// TIA Portal V18 export
FUNCTION_BLOCK "ST10_CountCycleTimeMain"   // FB1009, LAD
{ S7_Optimized_Access := 'TRUE' }
VERSION : 0.1
// stored: AutoNumber false, IsIECCheckEnabled false, IsRetainMemResEnabled false, MemoryReserve 100, SetENOAutomatically false, UDAEnableTagReadback false
   VAR_INPUT
      iAlwaysOn : Bool;
      iRun : Bool;
      iManualMode : Bool;
      iAutoMode : Bool;
      iAutoRunning : Bool;
   END_VAR
   VAR
      MianCountCycleTime { S7_SetPoint := 'True'} : "Count_CycleTime";
      PM1CountCycleTime { S7_SetPoint := 'True'} : "Count_CycleTime_V3";
      PM2CountCycleTime { S7_SetPoint := 'True'} : "Count_CycleTime_V3";
      PM3CountCycleTime { S7_SetPoint := 'True'} : "Count_CycleTime_V3";
      PM4CountCycleTime { S7_SetPoint := 'True'} : "Count_CycleTime_V3";
      PM5CountCycleTime { S7_SetPoint := 'True'} : "Count_CycleTime_V3";
      PM6CountCycleTime { S7_SetPoint := 'True'} : "Count_CycleTime_V3";
      PM7CountCycleTime { S7_SetPoint := 'True'} : "Count_CycleTime_V3";
      PM8CountCycleTime { S7_SetPoint := 'True'} : "Count_CycleTime_V3";
      PM9CountCycleTime { S7_SetPoint := 'True'} : "Count_CycleTime_V3";
      PM10CountCycleTime { S7_SetPoint := 'True'} : "Count_CycleTime_V3";
      PM11CountCycleTime { S7_SetPoint := 'True'} : "Count_CycleTime_V3";
      PM12CountCycleTime { S7_SetPoint := 'True'} : "Count_CycleTime_V3";
      PM13CountCycleTime { S7_SetPoint := 'True'} : "Count_CycleTime_V3";
      PM14CountCycleTime { S7_SetPoint := 'True'} : "Count_CycleTime_V3";
      PM15CountCycleTime { S7_SetPoint := 'True'} : "Count_CycleTime_V3";
      PM16CountCycleTime { S7_SetPoint := 'True'} : "Count_CycleTime_V3";
      PM17CountCycleTime { S7_SetPoint := 'True'} : "Count_CycleTime_V3";
      PM18CountCycleTime { S7_SetPoint := 'True'} : "Count_CycleTime_V3";
      PM19CountCycleTime { S7_SetPoint := 'True'} : "Count_CycleTime_V3";
      PM20CountCycleTime { S7_SetPoint := 'True'} : "Count_CycleTime_V3";
      PM21CountCycleTime { S7_SetPoint := 'True'} : "Count_CycleTime_V3";
      PM22CountCycleTime { S7_SetPoint := 'True'} : "Count_CycleTime_V3";
      PM23CountCycleTime { S7_SetPoint := 'True'} : "Count_CycleTime_V3";
      PM24CountCycleTime { S7_SetPoint := 'True'} : "Count_CycleTime_V3";
      PM25CountCycleTime { S7_SetPoint := 'True'} : "Count_CycleTime_V3";
      PM26CountCycleTime { S7_SetPoint := 'True'} : "Count_CycleTime_V3";
      PM27CountCycleTime { S7_SetPoint := 'True'} : "Count_CycleTime_V3";
      PM28CountCycleTime { S7_SetPoint := 'True'} : "Count_CycleTime_V3";
      PM29CountCycleTime { S7_SetPoint := 'True'} : "Count_CycleTime_V3";
      PM30CountCycleTime { S7_SetPoint := 'True'} : "Count_CycleTime_V3";
   END_VAR
BEGIN

REGION Network 1: Mian Count & CycleTime
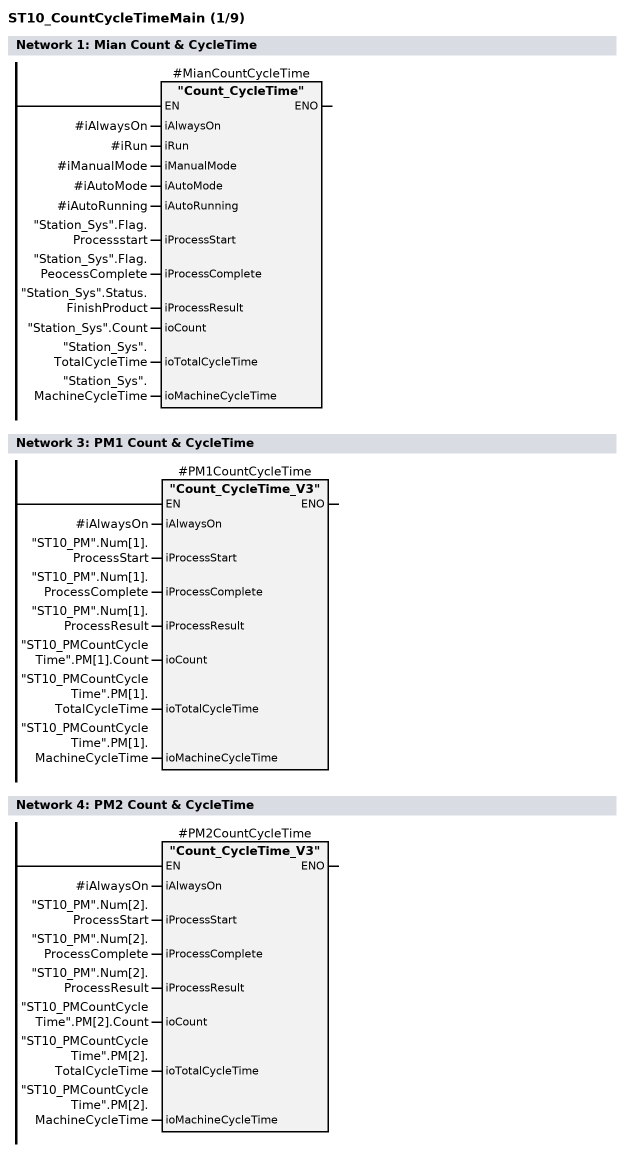
   RUNG wire#powerrail
      #MianCountCycleTime(iAlwaysOn := #iAlwaysOn, iRun := #iRun, iManualMode := #iManualMode, iAutoMode := #iAutoMode, iAutoRunning := #iAutoRunning, iProcessStart := "Station_Sys".Flag.Processstart, iProcessComplete := "Station_Sys".Flag.PeocessComplete, iProcessResult := "Station_Sys".Status.FinishProduct, ioCount := "Station_Sys".Count, ioTotalCycleTime := "Station_Sys".TotalCycleTime, ioMachineCycleTime := "Station_Sys".MachineCycleTime)
   END_RUNG
   // the same network as SCL:
   #MianCountCycleTime(iAlwaysOn := #iAlwaysOn,   // "Count_CycleTime"
                       iRun := #iRun,
                       iManualMode := #iManualMode,
                       iAutoMode := #iAutoMode,
                       iAutoRunning := #iAutoRunning,
                       iProcessStart := "Station_Sys".Flag.Processstart,
                       iProcessComplete := "Station_Sys".Flag.PeocessComplete,
                       iProcessResult := "Station_Sys".Status.FinishProduct,
                       ioCount := "Station_Sys".Count,
                       ioTotalCycleTime := "Station_Sys".TotalCycleTime,
                       ioMachineCycleTime := "Station_Sys".MachineCycleTime);
END_REGION

REGION Network 2 (SCL)
   "ST10_PMCountCycleTime".PM[1].Num := 1;
   "ST10_PMCountCycleTime".PM[2].Num := 2;
   "ST10_PMCountCycleTime".PM[3].Num := 3;
   "ST10_PMCountCycleTime".PM[4].Num := 4;
   "ST10_PMCountCycleTime".PM[5].Num := 5;
   "ST10_PMCountCycleTime".PM[6].Num := 6;
   "ST10_PMCountCycleTime".PM[7].Num := 7;
   "ST10_PMCountCycleTime".PM[8].Num := 8;
   "ST10_PMCountCycleTime".PM[9].Num := 9;
   "ST10_PMCountCycleTime".PM[10].Num := 10;
   "ST10_PMCountCycleTime".PM[11].Num := 11;
   "ST10_PMCountCycleTime".PM[12].Num := 12;
   "ST10_PMCountCycleTime".PM[13].Num := 13;
   "ST10_PMCountCycleTime".PM[14].Num := 14;
   "ST10_PMCountCycleTime".PM[15].Num := 15;
   "ST10_PMCountCycleTime".PM[16].Num := 16;
   "ST10_PMCountCycleTime".PM[17].Num := 17;
   "ST10_PMCountCycleTime".PM[18].Num := 18;
   "ST10_PMCountCycleTime".PM[19].Num := 19;
   "ST10_PMCountCycleTime".PM[20].Num := 20;
   "ST10_PMCountCycleTime".PM[21].Num := 21;
   "ST10_PMCountCycleTime".PM[22].Num := 22;
   "ST10_PMCountCycleTime".PM[23].Num := 23;
   "ST10_PMCountCycleTime".PM[24].Num := 24;
   "ST10_PMCountCycleTime".PM[25].Num := 25;
   // "ST70_PMCountCycleTime".PM[5].Num := 5;
   // "ST70_PMCountCycleTime".PM[6].Num := 6;
   // "ST70_PMCountCycleTime".PM[7].Num := 7;
   // "ST70_PMCountCycleTime".PM[8].Num := 8;
   // "ST70_PMCountCycleTime".PM[9].Num := 9;
   // "ST70_PMCountCycleTime".PM[10].Num := 10;
   //TEST
   (*
   "ST10_PMCountCycleTime".PM[1].Count.OK[0] := 10;
   "ST10_PMCountCycleTime".PM[2].Count.OK[0] := 20;
   "ST10_PMCountCycleTime".PM[3].Count.OK[0] := 30;
   "ST10_PMCountCycleTime".PM[4].Count.OK[0] := 40;
   "ST10_PMCountCycleTime".PM[5].Count.OK[0] := 50;
   "ST10_PMCountCycleTime".PM[6].Count.OK[0] := 60;
   "ST10_PMCountCycleTime".PM[7].Count.OK[0] := 70;
   "ST10_PMCountCycleTime".PM[8].Count.OK[0] := 80;
   "ST10_PMCountCycleTime".PM[9].Count.OK[0] := 90;
   "ST10_PMCountCycleTime".PM[10].Count.OK[0] := 100;

   "ST10_PMCountCycleTime".PM[1].TotalCycleTime.No[0] := 100;
   "ST10_PMCountCycleTime".PM[2].TotalCycleTime.No[0] := 200;
   "ST10_PMCountCycleTime".PM[3].TotalCycleTime.No[0] := 300;
   "ST10_PMCountCycleTime".PM[4].TotalCycleTime.No[0] := 400;
   "ST10_PMCountCycleTime".PM[5].TotalCycleTime.No[0] := 500;
   "ST10_PMCountCycleTime".PM[6].TotalCycleTime.No[0] := 600;
   "ST10_PMCountCycleTime".PM[7].TotalCycleTime.No[0] := 700;
   "ST10_PMCountCycleTime".PM[8].TotalCycleTime.No[0] := 800;
   "ST10_PMCountCycleTime".PM[9].TotalCycleTime.No[0] := 900;
   "ST10_PMCountCycleTime".PM[10].TotalCycleTime.No[0] := 1000;

   "ST10_PMCountCycleTime".PM[1].MachineCycleTime.No[0] := 110;
   "ST10_PMCountCycleTime".PM[2].MachineCycleTime.No[0] := 220;
   "ST10_PMCountCycleTime".PM[3].MachineCycleTime.No[0] := 330;
   "ST10_PMCountCycleTime".PM[4].MachineCycleTime.No[0] := 440;
   "ST10_PMCountCycleTime".PM[5].MachineCycleTime.No[0] := 550;
   "ST10_PMCountCycleTime".PM[6].MachineCycleTime.No[0] := 660;
   "ST10_PMCountCycleTime".PM[7].MachineCycleTime.No[0] := 770;
   "ST10_PMCountCycleTime".PM[8].MachineCycleTime.No[0] := 880;
   "ST10_PMCountCycleTime".PM[9].MachineCycleTime.No[0] := 990;
   "ST10_PMCountCycleTime".PM[10].MachineCycleTime.No[0] := 1010;
   *)
END_REGION

REGION Network 3: PM1 Count & CycleTime
   RUNG wire#powerrail
      #PM1CountCycleTime(iAlwaysOn := #iAlwaysOn, iProcessStart := "ST10_PM".Num[1].ProcessStart, iProcessComplete := "ST10_PM".Num[1].ProcessComplete, iProcessResult := "ST10_PM".Num[1].ProcessResult, ioCount := "ST10_PMCountCycleTime".PM[1].Count, ioTotalCycleTime := "ST10_PMCountCycleTime".PM[1].TotalCycleTime, ioMachineCycleTime := "ST10_PMCountCycleTime".PM[1].MachineCycleTime)
   END_RUNG
   // the same network as SCL:
   #PM1CountCycleTime(iAlwaysOn := #iAlwaysOn,   // "Count_CycleTime_V3"
                      iProcessStart := "ST10_PM".Num[1].ProcessStart,
                      iProcessComplete := "ST10_PM".Num[1].ProcessComplete,
                      iProcessResult := "ST10_PM".Num[1].ProcessResult,
                      ioCount := "ST10_PMCountCycleTime".PM[1].Count,
                      ioTotalCycleTime := "ST10_PMCountCycleTime".PM[1].TotalCycleTime,
                      ioMachineCycleTime := "ST10_PMCountCycleTime".PM[1].MachineCycleTime);
END_REGION

REGION Network 4: PM2 Count & CycleTime
   RUNG wire#powerrail
      #PM2CountCycleTime(iAlwaysOn := #iAlwaysOn, iProcessStart := "ST10_PM".Num[2].ProcessStart, iProcessComplete := "ST10_PM".Num[2].ProcessComplete, iProcessResult := "ST10_PM".Num[2].ProcessResult, ioCount := "ST10_PMCountCycleTime".PM[2].Count, ioTotalCycleTime := "ST10_PMCountCycleTime".PM[2].TotalCycleTime, ioMachineCycleTime := "ST10_PMCountCycleTime".PM[2].MachineCycleTime)
   END_RUNG
   // the same network as SCL:
   #PM2CountCycleTime(iAlwaysOn := #iAlwaysOn,   // "Count_CycleTime_V3"
                      iProcessStart := "ST10_PM".Num[2].ProcessStart,
                      iProcessComplete := "ST10_PM".Num[2].ProcessComplete,
                      iProcessResult := "ST10_PM".Num[2].ProcessResult,
                      ioCount := "ST10_PMCountCycleTime".PM[2].Count,
                      ioTotalCycleTime := "ST10_PMCountCycleTime".PM[2].TotalCycleTime,
                      ioMachineCycleTime := "ST10_PMCountCycleTime".PM[2].MachineCycleTime);
END_REGION

REGION Network 5: PM3 Count & CycleTime
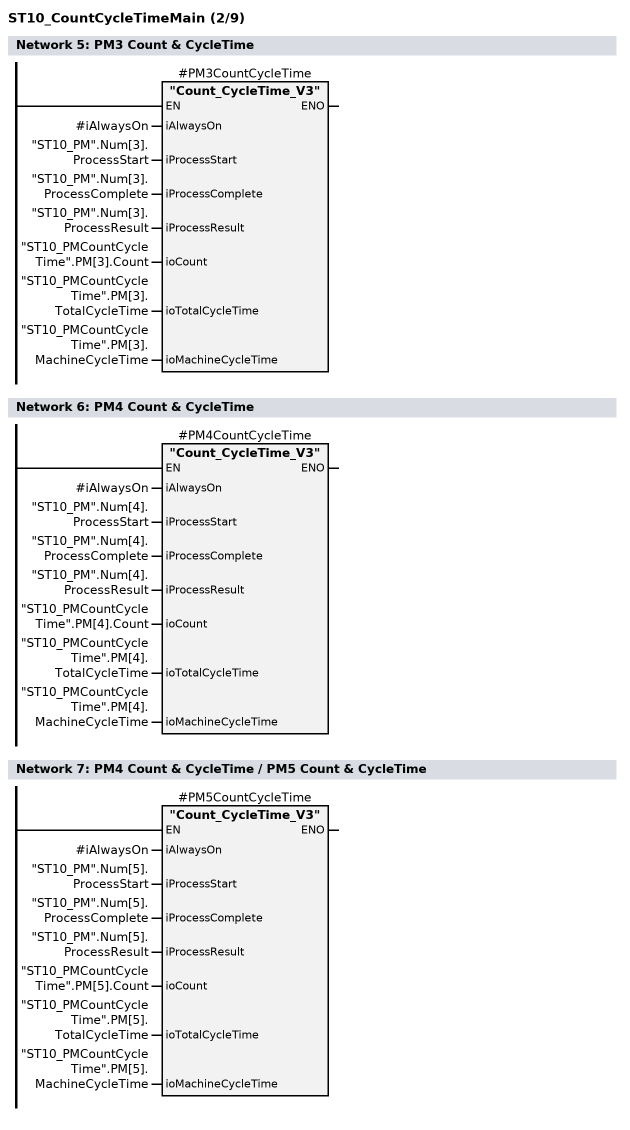
   RUNG wire#powerrail
      #PM3CountCycleTime(iAlwaysOn := #iAlwaysOn, iProcessStart := "ST10_PM".Num[3].ProcessStart, iProcessComplete := "ST10_PM".Num[3].ProcessComplete, iProcessResult := "ST10_PM".Num[3].ProcessResult, ioCount := "ST10_PMCountCycleTime".PM[3].Count, ioTotalCycleTime := "ST10_PMCountCycleTime".PM[3].TotalCycleTime, ioMachineCycleTime := "ST10_PMCountCycleTime".PM[3].MachineCycleTime)
   END_RUNG
   // the same network as SCL:
   #PM3CountCycleTime(iAlwaysOn := #iAlwaysOn,   // "Count_CycleTime_V3"
                      iProcessStart := "ST10_PM".Num[3].ProcessStart,
                      iProcessComplete := "ST10_PM".Num[3].ProcessComplete,
                      iProcessResult := "ST10_PM".Num[3].ProcessResult,
                      ioCount := "ST10_PMCountCycleTime".PM[3].Count,
                      ioTotalCycleTime := "ST10_PMCountCycleTime".PM[3].TotalCycleTime,
                      ioMachineCycleTime := "ST10_PMCountCycleTime".PM[3].MachineCycleTime);
END_REGION

REGION Network 6: PM4 Count & CycleTime
   RUNG wire#powerrail
      #PM4CountCycleTime(iAlwaysOn := #iAlwaysOn, iProcessStart := "ST10_PM".Num[4].ProcessStart, iProcessComplete := "ST10_PM".Num[4].ProcessComplete, iProcessResult := "ST10_PM".Num[4].ProcessResult, ioCount := "ST10_PMCountCycleTime".PM[4].Count, ioTotalCycleTime := "ST10_PMCountCycleTime".PM[4].TotalCycleTime, ioMachineCycleTime := "ST10_PMCountCycleTime".PM[4].MachineCycleTime)
   END_RUNG
   // the same network as SCL:
   #PM4CountCycleTime(iAlwaysOn := #iAlwaysOn,   // "Count_CycleTime_V3"
                      iProcessStart := "ST10_PM".Num[4].ProcessStart,
                      iProcessComplete := "ST10_PM".Num[4].ProcessComplete,
                      iProcessResult := "ST10_PM".Num[4].ProcessResult,
                      ioCount := "ST10_PMCountCycleTime".PM[4].Count,
                      ioTotalCycleTime := "ST10_PMCountCycleTime".PM[4].TotalCycleTime,
                      ioMachineCycleTime := "ST10_PMCountCycleTime".PM[4].MachineCycleTime);
END_REGION

REGION Network 7: PM4 Count & CycleTime / PM5 Count & CycleTime
   RUNG wire#powerrail
      #PM5CountCycleTime(iAlwaysOn := #iAlwaysOn, iProcessStart := "ST10_PM".Num[5].ProcessStart, iProcessComplete := "ST10_PM".Num[5].ProcessComplete, iProcessResult := "ST10_PM".Num[5].ProcessResult, ioCount := "ST10_PMCountCycleTime".PM[5].Count, ioTotalCycleTime := "ST10_PMCountCycleTime".PM[5].TotalCycleTime, ioMachineCycleTime := "ST10_PMCountCycleTime".PM[5].MachineCycleTime)
   END_RUNG
   // the same network as SCL:
   #PM5CountCycleTime(iAlwaysOn := #iAlwaysOn,   // "Count_CycleTime_V3"
                      iProcessStart := "ST10_PM".Num[5].ProcessStart,
                      iProcessComplete := "ST10_PM".Num[5].ProcessComplete,
                      iProcessResult := "ST10_PM".Num[5].ProcessResult,
                      ioCount := "ST10_PMCountCycleTime".PM[5].Count,
                      ioTotalCycleTime := "ST10_PMCountCycleTime".PM[5].TotalCycleTime,
                      ioMachineCycleTime := "ST10_PMCountCycleTime".PM[5].MachineCycleTime);
END_REGION

REGION Network 8: PM4 Count & CycleTime / PM6 Count & CycleTime
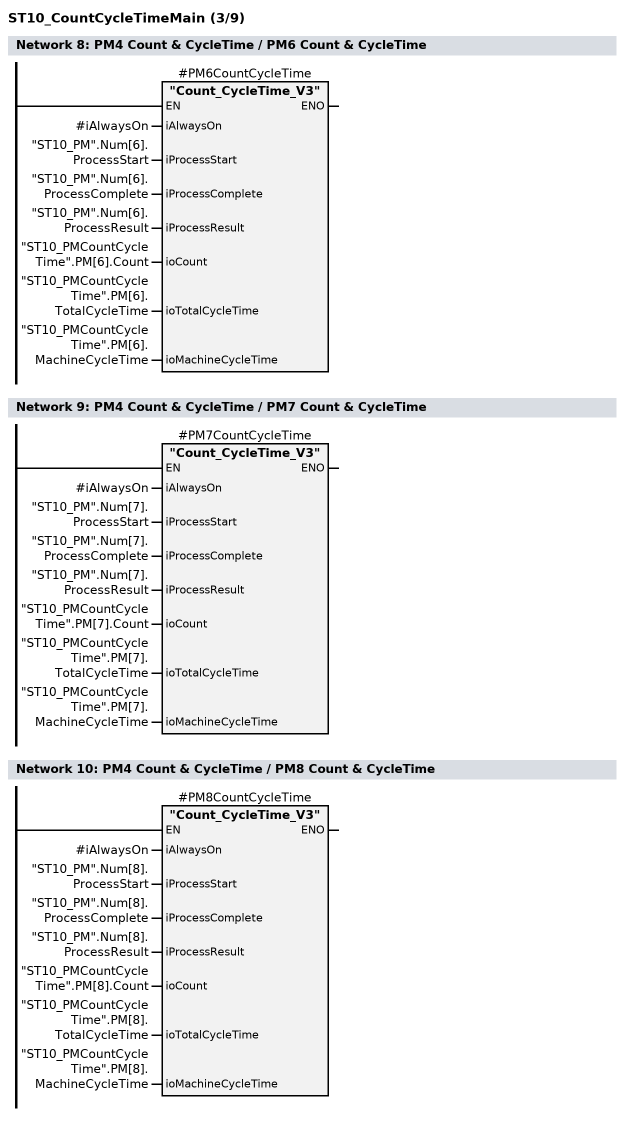
   RUNG wire#powerrail
      #PM6CountCycleTime(iAlwaysOn := #iAlwaysOn, iProcessStart := "ST10_PM".Num[6].ProcessStart, iProcessComplete := "ST10_PM".Num[6].ProcessComplete, iProcessResult := "ST10_PM".Num[6].ProcessResult, ioCount := "ST10_PMCountCycleTime".PM[6].Count, ioTotalCycleTime := "ST10_PMCountCycleTime".PM[6].TotalCycleTime, ioMachineCycleTime := "ST10_PMCountCycleTime".PM[6].MachineCycleTime)
   END_RUNG
   // the same network as SCL:
   #PM6CountCycleTime(iAlwaysOn := #iAlwaysOn,   // "Count_CycleTime_V3"
                      iProcessStart := "ST10_PM".Num[6].ProcessStart,
                      iProcessComplete := "ST10_PM".Num[6].ProcessComplete,
                      iProcessResult := "ST10_PM".Num[6].ProcessResult,
                      ioCount := "ST10_PMCountCycleTime".PM[6].Count,
                      ioTotalCycleTime := "ST10_PMCountCycleTime".PM[6].TotalCycleTime,
                      ioMachineCycleTime := "ST10_PMCountCycleTime".PM[6].MachineCycleTime);
END_REGION

REGION Network 9: PM4 Count & CycleTime / PM7 Count & CycleTime
   RUNG wire#powerrail
      #PM7CountCycleTime(iAlwaysOn := #iAlwaysOn, iProcessStart := "ST10_PM".Num[7].ProcessStart, iProcessComplete := "ST10_PM".Num[7].ProcessComplete, iProcessResult := "ST10_PM".Num[7].ProcessResult, ioCount := "ST10_PMCountCycleTime".PM[7].Count, ioTotalCycleTime := "ST10_PMCountCycleTime".PM[7].TotalCycleTime, ioMachineCycleTime := "ST10_PMCountCycleTime".PM[7].MachineCycleTime)
   END_RUNG
   // the same network as SCL:
   #PM7CountCycleTime(iAlwaysOn := #iAlwaysOn,   // "Count_CycleTime_V3"
                      iProcessStart := "ST10_PM".Num[7].ProcessStart,
                      iProcessComplete := "ST10_PM".Num[7].ProcessComplete,
                      iProcessResult := "ST10_PM".Num[7].ProcessResult,
                      ioCount := "ST10_PMCountCycleTime".PM[7].Count,
                      ioTotalCycleTime := "ST10_PMCountCycleTime".PM[7].TotalCycleTime,
                      ioMachineCycleTime := "ST10_PMCountCycleTime".PM[7].MachineCycleTime);
END_REGION

REGION Network 10: PM4 Count & CycleTime / PM8 Count & CycleTime
   RUNG wire#powerrail
      #PM8CountCycleTime(iAlwaysOn := #iAlwaysOn, iProcessStart := "ST10_PM".Num[8].ProcessStart, iProcessComplete := "ST10_PM".Num[8].ProcessComplete, iProcessResult := "ST10_PM".Num[8].ProcessResult, ioCount := "ST10_PMCountCycleTime".PM[8].Count, ioTotalCycleTime := "ST10_PMCountCycleTime".PM[8].TotalCycleTime, ioMachineCycleTime := "ST10_PMCountCycleTime".PM[8].MachineCycleTime)
   END_RUNG
   // the same network as SCL:
   #PM8CountCycleTime(iAlwaysOn := #iAlwaysOn,   // "Count_CycleTime_V3"
                      iProcessStart := "ST10_PM".Num[8].ProcessStart,
                      iProcessComplete := "ST10_PM".Num[8].ProcessComplete,
                      iProcessResult := "ST10_PM".Num[8].ProcessResult,
                      ioCount := "ST10_PMCountCycleTime".PM[8].Count,
                      ioTotalCycleTime := "ST10_PMCountCycleTime".PM[8].TotalCycleTime,
                      ioMachineCycleTime := "ST10_PMCountCycleTime".PM[8].MachineCycleTime);
END_REGION

REGION Network 11: PM4 Count & CycleTime / PM9 Count & CycleTime
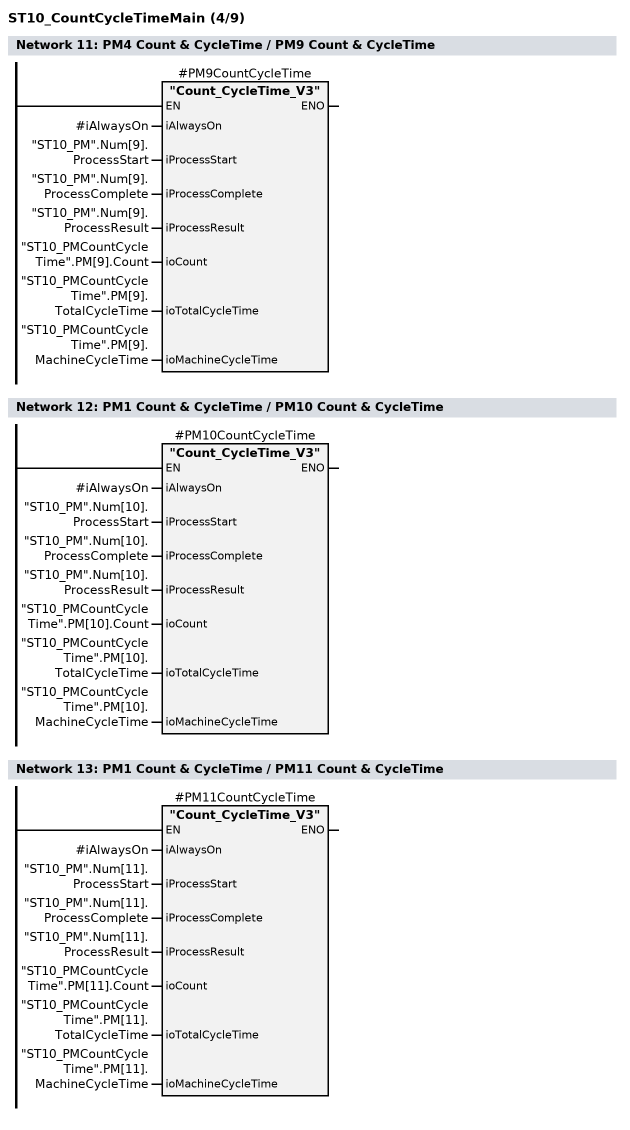
   RUNG wire#powerrail
      #PM9CountCycleTime(iAlwaysOn := #iAlwaysOn, iProcessStart := "ST10_PM".Num[9].ProcessStart, iProcessComplete := "ST10_PM".Num[9].ProcessComplete, iProcessResult := "ST10_PM".Num[9].ProcessResult, ioCount := "ST10_PMCountCycleTime".PM[9].Count, ioTotalCycleTime := "ST10_PMCountCycleTime".PM[9].TotalCycleTime, ioMachineCycleTime := "ST10_PMCountCycleTime".PM[9].MachineCycleTime)
   END_RUNG
   // the same network as SCL:
   #PM9CountCycleTime(iAlwaysOn := #iAlwaysOn,   // "Count_CycleTime_V3"
                      iProcessStart := "ST10_PM".Num[9].ProcessStart,
                      iProcessComplete := "ST10_PM".Num[9].ProcessComplete,
                      iProcessResult := "ST10_PM".Num[9].ProcessResult,
                      ioCount := "ST10_PMCountCycleTime".PM[9].Count,
                      ioTotalCycleTime := "ST10_PMCountCycleTime".PM[9].TotalCycleTime,
                      ioMachineCycleTime := "ST10_PMCountCycleTime".PM[9].MachineCycleTime);
END_REGION

REGION Network 12: PM1 Count & CycleTime / PM10 Count & CycleTime
   RUNG wire#powerrail
      #PM10CountCycleTime(iAlwaysOn := #iAlwaysOn, iProcessStart := "ST10_PM".Num[10].ProcessStart, iProcessComplete := "ST10_PM".Num[10].ProcessComplete, iProcessResult := "ST10_PM".Num[10].ProcessResult, ioCount := "ST10_PMCountCycleTime".PM[10].Count, ioTotalCycleTime := "ST10_PMCountCycleTime".PM[10].TotalCycleTime, ioMachineCycleTime := "ST10_PMCountCycleTime".PM[10].MachineCycleTime)
   END_RUNG
   // the same network as SCL:
   #PM10CountCycleTime(iAlwaysOn := #iAlwaysOn,   // "Count_CycleTime_V3"
                       iProcessStart := "ST10_PM".Num[10].ProcessStart,
                       iProcessComplete := "ST10_PM".Num[10].ProcessComplete,
                       iProcessResult := "ST10_PM".Num[10].ProcessResult,
                       ioCount := "ST10_PMCountCycleTime".PM[10].Count,
                       ioTotalCycleTime := "ST10_PMCountCycleTime".PM[10].TotalCycleTime,
                       ioMachineCycleTime := "ST10_PMCountCycleTime".PM[10].MachineCycleTime);
END_REGION

REGION Network 13: PM1 Count & CycleTime / PM11 Count & CycleTime
   RUNG wire#powerrail
      #PM11CountCycleTime(iAlwaysOn := #iAlwaysOn, iProcessStart := "ST10_PM".Num[11].ProcessStart, iProcessComplete := "ST10_PM".Num[11].ProcessComplete, iProcessResult := "ST10_PM".Num[11].ProcessResult, ioCount := "ST10_PMCountCycleTime".PM[11].Count, ioTotalCycleTime := "ST10_PMCountCycleTime".PM[11].TotalCycleTime, ioMachineCycleTime := "ST10_PMCountCycleTime".PM[11].MachineCycleTime)
   END_RUNG
   // the same network as SCL:
   #PM11CountCycleTime(iAlwaysOn := #iAlwaysOn,   // "Count_CycleTime_V3"
                       iProcessStart := "ST10_PM".Num[11].ProcessStart,
                       iProcessComplete := "ST10_PM".Num[11].ProcessComplete,
                       iProcessResult := "ST10_PM".Num[11].ProcessResult,
                       ioCount := "ST10_PMCountCycleTime".PM[11].Count,
                       ioTotalCycleTime := "ST10_PMCountCycleTime".PM[11].TotalCycleTime,
                       ioMachineCycleTime := "ST10_PMCountCycleTime".PM[11].MachineCycleTime);
END_REGION

REGION Network 14: PM1 Count & CycleTime / PM12 Count & CycleTime
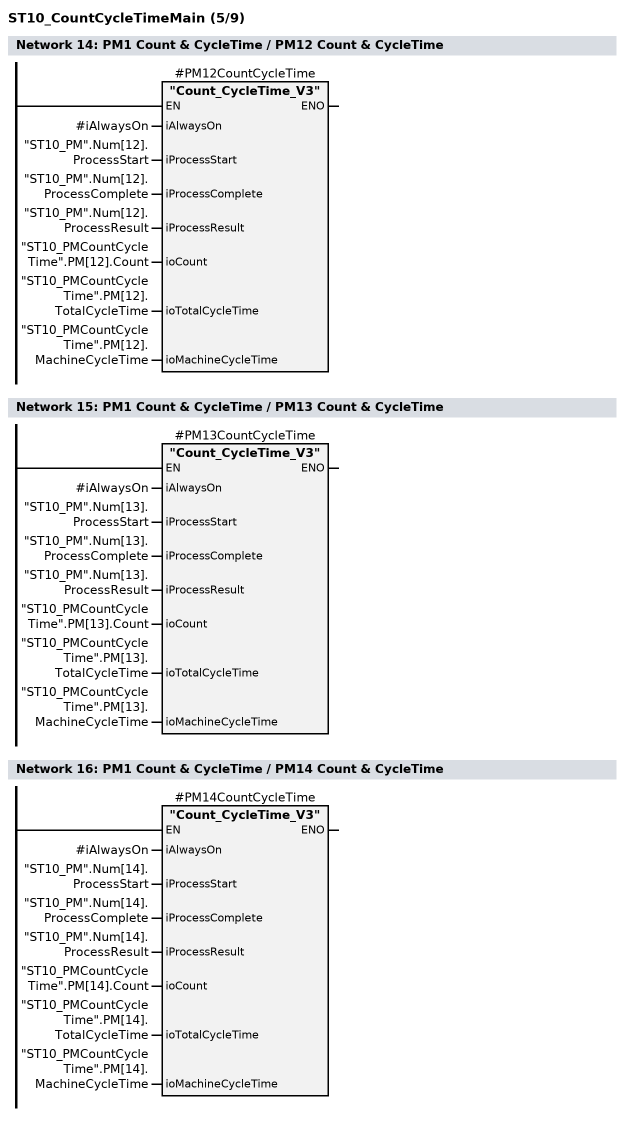
   RUNG wire#powerrail
      #PM12CountCycleTime(iAlwaysOn := #iAlwaysOn, iProcessStart := "ST10_PM".Num[12].ProcessStart, iProcessComplete := "ST10_PM".Num[12].ProcessComplete, iProcessResult := "ST10_PM".Num[12].ProcessResult, ioCount := "ST10_PMCountCycleTime".PM[12].Count, ioTotalCycleTime := "ST10_PMCountCycleTime".PM[12].TotalCycleTime, ioMachineCycleTime := "ST10_PMCountCycleTime".PM[12].MachineCycleTime)
   END_RUNG
   // the same network as SCL:
   #PM12CountCycleTime(iAlwaysOn := #iAlwaysOn,   // "Count_CycleTime_V3"
                       iProcessStart := "ST10_PM".Num[12].ProcessStart,
                       iProcessComplete := "ST10_PM".Num[12].ProcessComplete,
                       iProcessResult := "ST10_PM".Num[12].ProcessResult,
                       ioCount := "ST10_PMCountCycleTime".PM[12].Count,
                       ioTotalCycleTime := "ST10_PMCountCycleTime".PM[12].TotalCycleTime,
                       ioMachineCycleTime := "ST10_PMCountCycleTime".PM[12].MachineCycleTime);
END_REGION

REGION Network 15: PM1 Count & CycleTime / PM13 Count & CycleTime
   RUNG wire#powerrail
      #PM13CountCycleTime(iAlwaysOn := #iAlwaysOn, iProcessStart := "ST10_PM".Num[13].ProcessStart, iProcessComplete := "ST10_PM".Num[13].ProcessComplete, iProcessResult := "ST10_PM".Num[13].ProcessResult, ioCount := "ST10_PMCountCycleTime".PM[13].Count, ioTotalCycleTime := "ST10_PMCountCycleTime".PM[13].TotalCycleTime, ioMachineCycleTime := "ST10_PMCountCycleTime".PM[13].MachineCycleTime)
   END_RUNG
   // the same network as SCL:
   #PM13CountCycleTime(iAlwaysOn := #iAlwaysOn,   // "Count_CycleTime_V3"
                       iProcessStart := "ST10_PM".Num[13].ProcessStart,
                       iProcessComplete := "ST10_PM".Num[13].ProcessComplete,
                       iProcessResult := "ST10_PM".Num[13].ProcessResult,
                       ioCount := "ST10_PMCountCycleTime".PM[13].Count,
                       ioTotalCycleTime := "ST10_PMCountCycleTime".PM[13].TotalCycleTime,
                       ioMachineCycleTime := "ST10_PMCountCycleTime".PM[13].MachineCycleTime);
END_REGION

REGION Network 16: PM1 Count & CycleTime / PM14 Count & CycleTime
   RUNG wire#powerrail
      #PM14CountCycleTime(iAlwaysOn := #iAlwaysOn, iProcessStart := "ST10_PM".Num[14].ProcessStart, iProcessComplete := "ST10_PM".Num[14].ProcessComplete, iProcessResult := "ST10_PM".Num[14].ProcessResult, ioCount := "ST10_PMCountCycleTime".PM[14].Count, ioTotalCycleTime := "ST10_PMCountCycleTime".PM[14].TotalCycleTime, ioMachineCycleTime := "ST10_PMCountCycleTime".PM[14].MachineCycleTime)
   END_RUNG
   // the same network as SCL:
   #PM14CountCycleTime(iAlwaysOn := #iAlwaysOn,   // "Count_CycleTime_V3"
                       iProcessStart := "ST10_PM".Num[14].ProcessStart,
                       iProcessComplete := "ST10_PM".Num[14].ProcessComplete,
                       iProcessResult := "ST10_PM".Num[14].ProcessResult,
                       ioCount := "ST10_PMCountCycleTime".PM[14].Count,
                       ioTotalCycleTime := "ST10_PMCountCycleTime".PM[14].TotalCycleTime,
                       ioMachineCycleTime := "ST10_PMCountCycleTime".PM[14].MachineCycleTime);
END_REGION

REGION Network 17: PM1 Count & CycleTime / PM15 Count & CycleTime
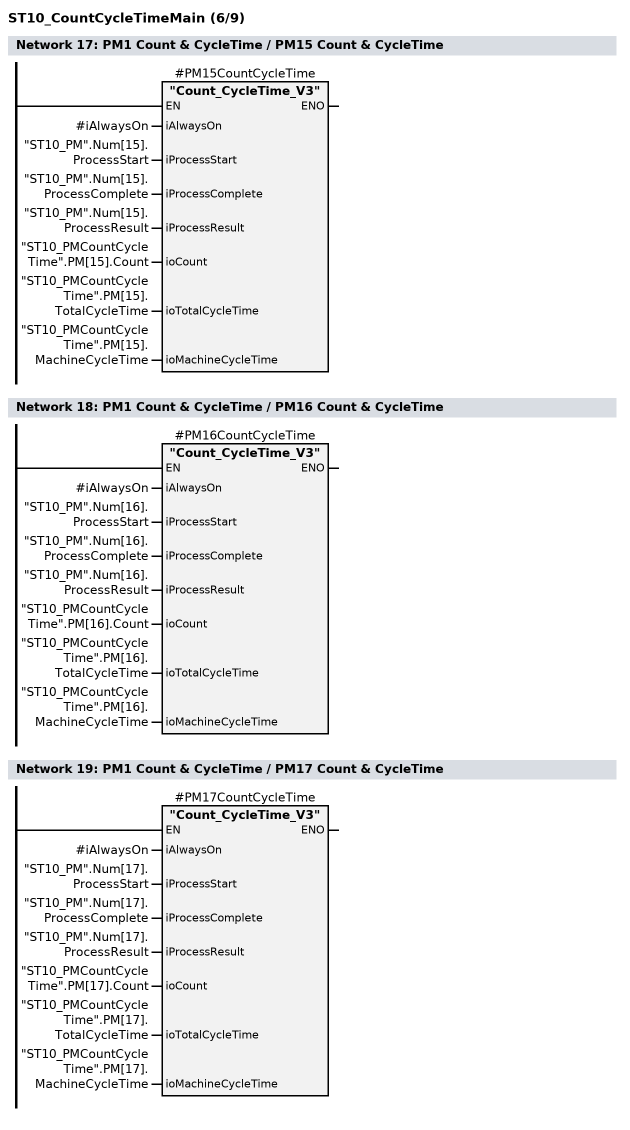
   RUNG wire#powerrail
      #PM15CountCycleTime(iAlwaysOn := #iAlwaysOn, iProcessStart := "ST10_PM".Num[15].ProcessStart, iProcessComplete := "ST10_PM".Num[15].ProcessComplete, iProcessResult := "ST10_PM".Num[15].ProcessResult, ioCount := "ST10_PMCountCycleTime".PM[15].Count, ioTotalCycleTime := "ST10_PMCountCycleTime".PM[15].TotalCycleTime, ioMachineCycleTime := "ST10_PMCountCycleTime".PM[15].MachineCycleTime)
   END_RUNG
   // the same network as SCL:
   #PM15CountCycleTime(iAlwaysOn := #iAlwaysOn,   // "Count_CycleTime_V3"
                       iProcessStart := "ST10_PM".Num[15].ProcessStart,
                       iProcessComplete := "ST10_PM".Num[15].ProcessComplete,
                       iProcessResult := "ST10_PM".Num[15].ProcessResult,
                       ioCount := "ST10_PMCountCycleTime".PM[15].Count,
                       ioTotalCycleTime := "ST10_PMCountCycleTime".PM[15].TotalCycleTime,
                       ioMachineCycleTime := "ST10_PMCountCycleTime".PM[15].MachineCycleTime);
END_REGION

REGION Network 18: PM1 Count & CycleTime / PM16 Count & CycleTime
   RUNG wire#powerrail
      #PM16CountCycleTime(iAlwaysOn := #iAlwaysOn, iProcessStart := "ST10_PM".Num[16].ProcessStart, iProcessComplete := "ST10_PM".Num[16].ProcessComplete, iProcessResult := "ST10_PM".Num[16].ProcessResult, ioCount := "ST10_PMCountCycleTime".PM[16].Count, ioTotalCycleTime := "ST10_PMCountCycleTime".PM[16].TotalCycleTime, ioMachineCycleTime := "ST10_PMCountCycleTime".PM[16].MachineCycleTime)
   END_RUNG
   // the same network as SCL:
   #PM16CountCycleTime(iAlwaysOn := #iAlwaysOn,   // "Count_CycleTime_V3"
                       iProcessStart := "ST10_PM".Num[16].ProcessStart,
                       iProcessComplete := "ST10_PM".Num[16].ProcessComplete,
                       iProcessResult := "ST10_PM".Num[16].ProcessResult,
                       ioCount := "ST10_PMCountCycleTime".PM[16].Count,
                       ioTotalCycleTime := "ST10_PMCountCycleTime".PM[16].TotalCycleTime,
                       ioMachineCycleTime := "ST10_PMCountCycleTime".PM[16].MachineCycleTime);
END_REGION

REGION Network 19: PM1 Count & CycleTime / PM17 Count & CycleTime
   RUNG wire#powerrail
      #PM17CountCycleTime(iAlwaysOn := #iAlwaysOn, iProcessStart := "ST10_PM".Num[17].ProcessStart, iProcessComplete := "ST10_PM".Num[17].ProcessComplete, iProcessResult := "ST10_PM".Num[17].ProcessResult, ioCount := "ST10_PMCountCycleTime".PM[17].Count, ioTotalCycleTime := "ST10_PMCountCycleTime".PM[17].TotalCycleTime, ioMachineCycleTime := "ST10_PMCountCycleTime".PM[17].MachineCycleTime)
   END_RUNG
   // the same network as SCL:
   #PM17CountCycleTime(iAlwaysOn := #iAlwaysOn,   // "Count_CycleTime_V3"
                       iProcessStart := "ST10_PM".Num[17].ProcessStart,
                       iProcessComplete := "ST10_PM".Num[17].ProcessComplete,
                       iProcessResult := "ST10_PM".Num[17].ProcessResult,
                       ioCount := "ST10_PMCountCycleTime".PM[17].Count,
                       ioTotalCycleTime := "ST10_PMCountCycleTime".PM[17].TotalCycleTime,
                       ioMachineCycleTime := "ST10_PMCountCycleTime".PM[17].MachineCycleTime);
END_REGION

REGION Network 20: PM1 Count & CycleTime / PM18 Count & CycleTime
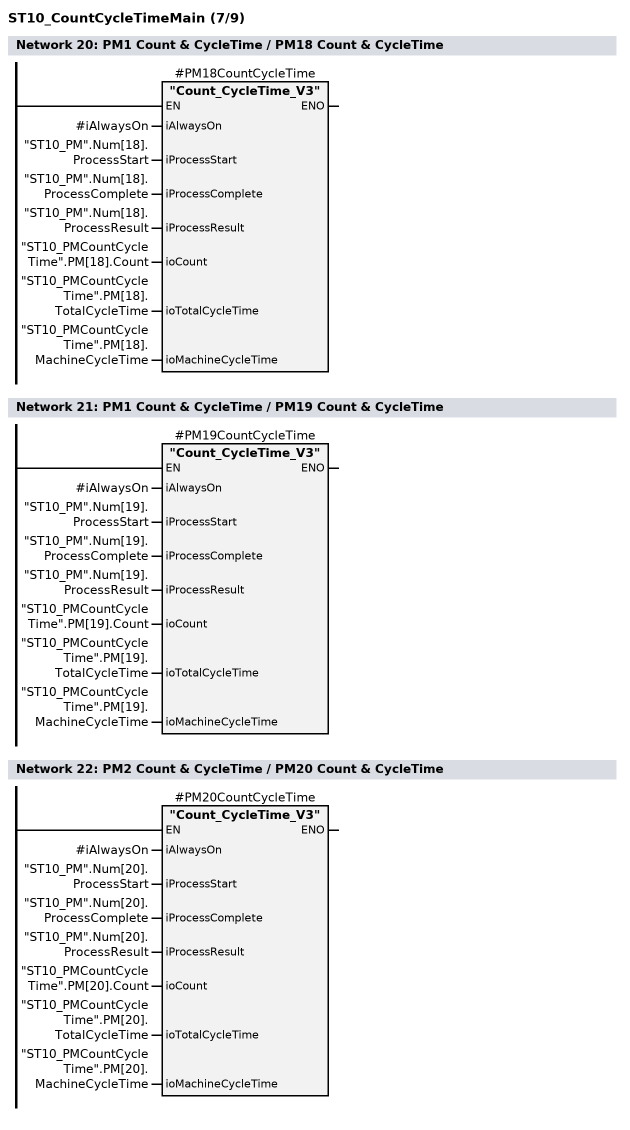
   RUNG wire#powerrail
      #PM18CountCycleTime(iAlwaysOn := #iAlwaysOn, iProcessStart := "ST10_PM".Num[18].ProcessStart, iProcessComplete := "ST10_PM".Num[18].ProcessComplete, iProcessResult := "ST10_PM".Num[18].ProcessResult, ioCount := "ST10_PMCountCycleTime".PM[18].Count, ioTotalCycleTime := "ST10_PMCountCycleTime".PM[18].TotalCycleTime, ioMachineCycleTime := "ST10_PMCountCycleTime".PM[18].MachineCycleTime)
   END_RUNG
   // the same network as SCL:
   #PM18CountCycleTime(iAlwaysOn := #iAlwaysOn,   // "Count_CycleTime_V3"
                       iProcessStart := "ST10_PM".Num[18].ProcessStart,
                       iProcessComplete := "ST10_PM".Num[18].ProcessComplete,
                       iProcessResult := "ST10_PM".Num[18].ProcessResult,
                       ioCount := "ST10_PMCountCycleTime".PM[18].Count,
                       ioTotalCycleTime := "ST10_PMCountCycleTime".PM[18].TotalCycleTime,
                       ioMachineCycleTime := "ST10_PMCountCycleTime".PM[18].MachineCycleTime);
END_REGION

REGION Network 21: PM1 Count & CycleTime / PM19 Count & CycleTime
   RUNG wire#powerrail
      #PM19CountCycleTime(iAlwaysOn := #iAlwaysOn, iProcessStart := "ST10_PM".Num[19].ProcessStart, iProcessComplete := "ST10_PM".Num[19].ProcessComplete, iProcessResult := "ST10_PM".Num[19].ProcessResult, ioCount := "ST10_PMCountCycleTime".PM[19].Count, ioTotalCycleTime := "ST10_PMCountCycleTime".PM[19].TotalCycleTime, ioMachineCycleTime := "ST10_PMCountCycleTime".PM[19].MachineCycleTime)
   END_RUNG
   // the same network as SCL:
   #PM19CountCycleTime(iAlwaysOn := #iAlwaysOn,   // "Count_CycleTime_V3"
                       iProcessStart := "ST10_PM".Num[19].ProcessStart,
                       iProcessComplete := "ST10_PM".Num[19].ProcessComplete,
                       iProcessResult := "ST10_PM".Num[19].ProcessResult,
                       ioCount := "ST10_PMCountCycleTime".PM[19].Count,
                       ioTotalCycleTime := "ST10_PMCountCycleTime".PM[19].TotalCycleTime,
                       ioMachineCycleTime := "ST10_PMCountCycleTime".PM[19].MachineCycleTime);
END_REGION

REGION Network 22: PM2 Count & CycleTime / PM20 Count & CycleTime
   RUNG wire#powerrail
      #PM20CountCycleTime(iAlwaysOn := #iAlwaysOn, iProcessStart := "ST10_PM".Num[20].ProcessStart, iProcessComplete := "ST10_PM".Num[20].ProcessComplete, iProcessResult := "ST10_PM".Num[20].ProcessResult, ioCount := "ST10_PMCountCycleTime".PM[20].Count, ioTotalCycleTime := "ST10_PMCountCycleTime".PM[20].TotalCycleTime, ioMachineCycleTime := "ST10_PMCountCycleTime".PM[20].MachineCycleTime)
   END_RUNG
   // the same network as SCL:
   #PM20CountCycleTime(iAlwaysOn := #iAlwaysOn,   // "Count_CycleTime_V3"
                       iProcessStart := "ST10_PM".Num[20].ProcessStart,
                       iProcessComplete := "ST10_PM".Num[20].ProcessComplete,
                       iProcessResult := "ST10_PM".Num[20].ProcessResult,
                       ioCount := "ST10_PMCountCycleTime".PM[20].Count,
                       ioTotalCycleTime := "ST10_PMCountCycleTime".PM[20].TotalCycleTime,
                       ioMachineCycleTime := "ST10_PMCountCycleTime".PM[20].MachineCycleTime);
END_REGION

REGION Network 23: PM2 Count & CycleTime / PM21 Count & CycleTime
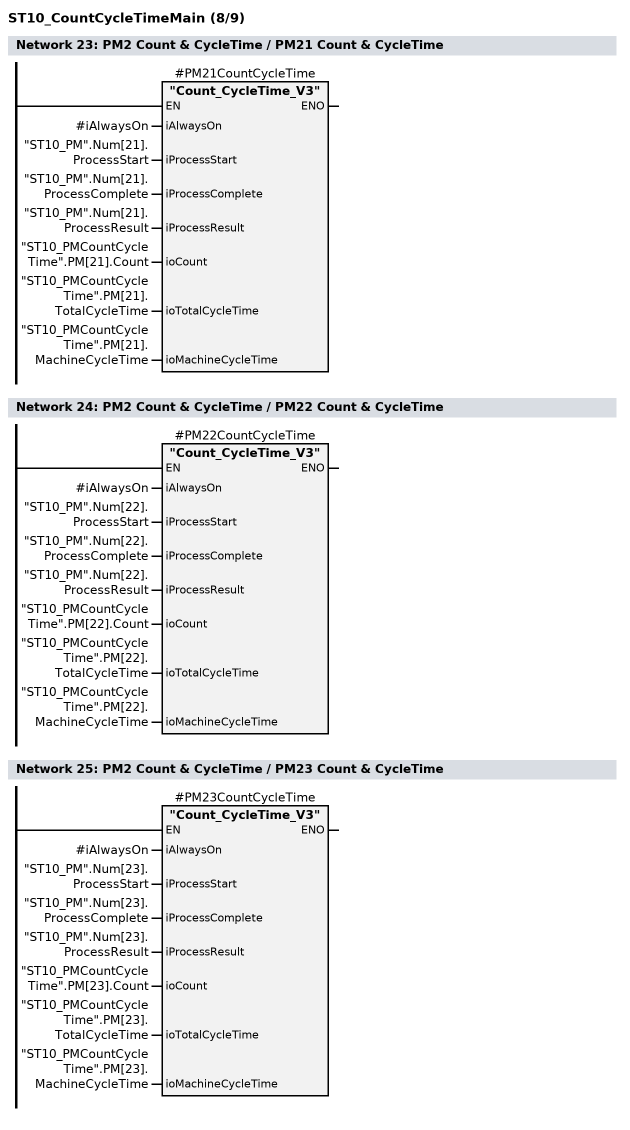
   RUNG wire#powerrail
      #PM21CountCycleTime(iAlwaysOn := #iAlwaysOn, iProcessStart := "ST10_PM".Num[21].ProcessStart, iProcessComplete := "ST10_PM".Num[21].ProcessComplete, iProcessResult := "ST10_PM".Num[21].ProcessResult, ioCount := "ST10_PMCountCycleTime".PM[21].Count, ioTotalCycleTime := "ST10_PMCountCycleTime".PM[21].TotalCycleTime, ioMachineCycleTime := "ST10_PMCountCycleTime".PM[21].MachineCycleTime)
   END_RUNG
   // the same network as SCL:
   #PM21CountCycleTime(iAlwaysOn := #iAlwaysOn,   // "Count_CycleTime_V3"
                       iProcessStart := "ST10_PM".Num[21].ProcessStart,
                       iProcessComplete := "ST10_PM".Num[21].ProcessComplete,
                       iProcessResult := "ST10_PM".Num[21].ProcessResult,
                       ioCount := "ST10_PMCountCycleTime".PM[21].Count,
                       ioTotalCycleTime := "ST10_PMCountCycleTime".PM[21].TotalCycleTime,
                       ioMachineCycleTime := "ST10_PMCountCycleTime".PM[21].MachineCycleTime);
END_REGION

REGION Network 24: PM2 Count & CycleTime / PM22 Count & CycleTime
   RUNG wire#powerrail
      #PM22CountCycleTime(iAlwaysOn := #iAlwaysOn, iProcessStart := "ST10_PM".Num[22].ProcessStart, iProcessComplete := "ST10_PM".Num[22].ProcessComplete, iProcessResult := "ST10_PM".Num[22].ProcessResult, ioCount := "ST10_PMCountCycleTime".PM[22].Count, ioTotalCycleTime := "ST10_PMCountCycleTime".PM[22].TotalCycleTime, ioMachineCycleTime := "ST10_PMCountCycleTime".PM[22].MachineCycleTime)
   END_RUNG
   // the same network as SCL:
   #PM22CountCycleTime(iAlwaysOn := #iAlwaysOn,   // "Count_CycleTime_V3"
                       iProcessStart := "ST10_PM".Num[22].ProcessStart,
                       iProcessComplete := "ST10_PM".Num[22].ProcessComplete,
                       iProcessResult := "ST10_PM".Num[22].ProcessResult,
                       ioCount := "ST10_PMCountCycleTime".PM[22].Count,
                       ioTotalCycleTime := "ST10_PMCountCycleTime".PM[22].TotalCycleTime,
                       ioMachineCycleTime := "ST10_PMCountCycleTime".PM[22].MachineCycleTime);
END_REGION

REGION Network 25: PM2 Count & CycleTime / PM23 Count & CycleTime
   RUNG wire#powerrail
      #PM23CountCycleTime(iAlwaysOn := #iAlwaysOn, iProcessStart := "ST10_PM".Num[23].ProcessStart, iProcessComplete := "ST10_PM".Num[23].ProcessComplete, iProcessResult := "ST10_PM".Num[23].ProcessResult, ioCount := "ST10_PMCountCycleTime".PM[23].Count, ioTotalCycleTime := "ST10_PMCountCycleTime".PM[23].TotalCycleTime, ioMachineCycleTime := "ST10_PMCountCycleTime".PM[23].MachineCycleTime)
   END_RUNG
   // the same network as SCL:
   #PM23CountCycleTime(iAlwaysOn := #iAlwaysOn,   // "Count_CycleTime_V3"
                       iProcessStart := "ST10_PM".Num[23].ProcessStart,
                       iProcessComplete := "ST10_PM".Num[23].ProcessComplete,
                       iProcessResult := "ST10_PM".Num[23].ProcessResult,
                       ioCount := "ST10_PMCountCycleTime".PM[23].Count,
                       ioTotalCycleTime := "ST10_PMCountCycleTime".PM[23].TotalCycleTime,
                       ioMachineCycleTime := "ST10_PMCountCycleTime".PM[23].MachineCycleTime);
END_REGION

REGION Network 26: PM2 Count & CycleTime / PM24 Count & CycleTime
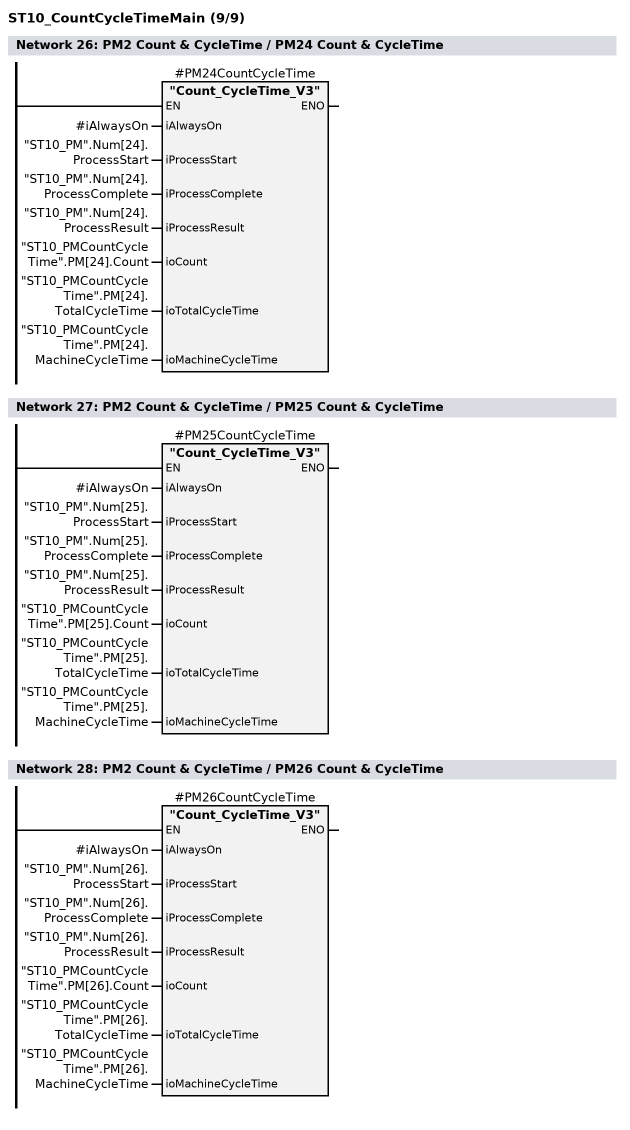
   RUNG wire#powerrail
      #PM24CountCycleTime(iAlwaysOn := #iAlwaysOn, iProcessStart := "ST10_PM".Num[24].ProcessStart, iProcessComplete := "ST10_PM".Num[24].ProcessComplete, iProcessResult := "ST10_PM".Num[24].ProcessResult, ioCount := "ST10_PMCountCycleTime".PM[24].Count, ioTotalCycleTime := "ST10_PMCountCycleTime".PM[24].TotalCycleTime, ioMachineCycleTime := "ST10_PMCountCycleTime".PM[24].MachineCycleTime)
   END_RUNG
   // the same network as SCL:
   #PM24CountCycleTime(iAlwaysOn := #iAlwaysOn,   // "Count_CycleTime_V3"
                       iProcessStart := "ST10_PM".Num[24].ProcessStart,
                       iProcessComplete := "ST10_PM".Num[24].ProcessComplete,
                       iProcessResult := "ST10_PM".Num[24].ProcessResult,
                       ioCount := "ST10_PMCountCycleTime".PM[24].Count,
                       ioTotalCycleTime := "ST10_PMCountCycleTime".PM[24].TotalCycleTime,
                       ioMachineCycleTime := "ST10_PMCountCycleTime".PM[24].MachineCycleTime);
END_REGION

REGION Network 27: PM2 Count & CycleTime / PM25 Count & CycleTime
   RUNG wire#powerrail
      #PM25CountCycleTime(iAlwaysOn := #iAlwaysOn, iProcessStart := "ST10_PM".Num[25].ProcessStart, iProcessComplete := "ST10_PM".Num[25].ProcessComplete, iProcessResult := "ST10_PM".Num[25].ProcessResult, ioCount := "ST10_PMCountCycleTime".PM[25].Count, ioTotalCycleTime := "ST10_PMCountCycleTime".PM[25].TotalCycleTime, ioMachineCycleTime := "ST10_PMCountCycleTime".PM[25].MachineCycleTime)
   END_RUNG
   // the same network as SCL:
   #PM25CountCycleTime(iAlwaysOn := #iAlwaysOn,   // "Count_CycleTime_V3"
                       iProcessStart := "ST10_PM".Num[25].ProcessStart,
                       iProcessComplete := "ST10_PM".Num[25].ProcessComplete,
                       iProcessResult := "ST10_PM".Num[25].ProcessResult,
                       ioCount := "ST10_PMCountCycleTime".PM[25].Count,
                       ioTotalCycleTime := "ST10_PMCountCycleTime".PM[25].TotalCycleTime,
                       ioMachineCycleTime := "ST10_PMCountCycleTime".PM[25].MachineCycleTime);
END_REGION

REGION Network 28: PM2 Count & CycleTime / PM26 Count & CycleTime
   RUNG wire#powerrail
      #PM26CountCycleTime(iAlwaysOn := #iAlwaysOn, iProcessStart := "ST10_PM".Num[26].ProcessStart, iProcessComplete := "ST10_PM".Num[26].ProcessComplete, iProcessResult := "ST10_PM".Num[26].ProcessResult, ioCount := "ST10_PMCountCycleTime".PM[26].Count, ioTotalCycleTime := "ST10_PMCountCycleTime".PM[26].TotalCycleTime, ioMachineCycleTime := "ST10_PMCountCycleTime".PM[26].MachineCycleTime)
   END_RUNG
   // the same network as SCL:
   #PM26CountCycleTime(iAlwaysOn := #iAlwaysOn,   // "Count_CycleTime_V3"
                       iProcessStart := "ST10_PM".Num[26].ProcessStart,
                       iProcessComplete := "ST10_PM".Num[26].ProcessComplete,
                       iProcessResult := "ST10_PM".Num[26].ProcessResult,
                       ioCount := "ST10_PMCountCycleTime".PM[26].Count,
                       ioTotalCycleTime := "ST10_PMCountCycleTime".PM[26].TotalCycleTime,
                       ioMachineCycleTime := "ST10_PMCountCycleTime".PM[26].MachineCycleTime);
END_REGION
END_FUNCTION_BLOCK
